(* PLC project LMM.project, Inovance company InoProShop(V1.9.1.6) InoProShop(V1.9.1.6) *)
(* stored: creationDateTime 2026-07-21T20:30:28.2051224, modificationDateTime 2026-07-21T19:55:23.2405761 *)

VAR_GLOBAL  (* GVL *)
  StartBtn AT %IX1.6 : BOOL;  (* 【面板启动】AT %IX1.6 → HMI_xStart/HMI_xEnable（上升沿 STOP→RUN） *)
  StopBtn AT %IX1.4 : BOOL;  (* 【面板停止】AT %IX1.4 → HMI_xStop *)
  ResetBtn : BOOL;  (* 【面板复位】→ HMI_xStopHold3s（错误复位脉冲）；地址现场可另绑 *)
  EStop AT %IX0.4 : BOOL;  (* 【面板急停】AT %IX0.4 正常=TRUE 按下=FALSE → 直通 HMI_xEStop *)
  StopLamp AT %QX0.6 : BOOL;  (* 【停止指示灯】AT %QX0.6 ← Dev_xStop（停止/待机） *)
  StartLamp AT %QX0.7 : BOOL;  (* 【启动/运行指示灯】AT %QX0.7 ← Dev_xRun（正在运行） *)
  JogVel : REAL;  (* 面板点动速度 → 桥接到 HMI_rJogVel* *)
  JogFwd : BOOL;  (* 面板前进 → 按 X 模式映射到 Sync/Diff/独立点动+ *)
  JogBwd : BOOL;  (* 面板后退 → 按 X 模式映射到 Sync/Diff/独立点动- *)
  JogUp : BOOL;  (* 面板上 → HMI_xJogZPos *)
  JogDown : BOOL;  (* 面板下 → HMI_xJogZNeg *)
  JogRight : BOOL;  (* 面板右 → HMI_xJogYPos *)
  JogLeft : BOOL;  (* 面板左 → HMI_xJogYNeg *)
  JogClockAdd : BOOL;  (* 顺时针 *)
  JogClockMis : BOOL;  (* 逆时针 *)
  JogACC : REAL;  (* 点动加速度 → AxisCmd_rAcc *)
  JogDEC : REAL;  (* 点动减速度 → AxisCmd_rDec *)
  HomeReq : BOOL;  (* 面板回零 → HMI_xHomeReqY/Z *)
  CaliForReq : BOOL;  (* 重力标定 *)
  ClearBruch : BOOL;  (* 毛刷清洗 *)
  yLength : REAL;  (* 龙门跨距/Y长度设定 4..6m → HMI_rWheelBase *)
  HMI_xEStop : BOOL;  (* 【急停】TRUE=未按下(正常)；FALSE=急停按下。可按可松，锁存由Logic保持 *)
  HMI_xStop : BOOL;  (* 【设备停止】短按RUN→STOP；长按3s故障复位 *)
  HMI_xStopHold3s : BOOL;  (* 【停止长按满3s脉冲】清急停锁存+轴错误复位+下使能 *)
  HMI_xEnable : BOOL;  (* 【使能/启动别名】与HMI_xStart等效；上升沿STOP→RUN *)
  Dev_xError : BOOL;  (* 【内部故障态】 *)
  Dev_xRun : BOOL;  (* 【内部运行态】 *)
  Dev_xStop : BOOL;  (* 【内部停机态】 *)
  eDevState : INT;  (* 【废弃】不做控制；显示请用 HMI_eDevState 派生 *)
  HMI_xDevError : BOOL;  (* 【故障灯设备级】 *)
  HMI_xDevRun : BOOL;  (* 【运行灯】 *)
  HMI_xDevStop : BOOL;  (* 【停机灯】 *)
  HMI_eOpMode : INT;  (* 【运行方式】0手动 1自动；配合Run灯 *)
  HMI_eDevState : INT;  (* 【设备状态码】0=STOP 1=RUN 2=ERROR *)
  HMI_xStart : BOOL;  (* 【设备启动】瞬时；上升沿STOP→RUN *)
  HMI_xJogYPos : BOOL;  (* 【Y点动+】TRUE移动 FALSE暂停；受限位/Z忙 *)
  HMI_xJogYNeg : BOOL;  (* 【Y点动-】TRUE移动 FALSE暂停 *)
  HMI_xJogZPos : BOOL;  (* 【Z点动+】TRUE移动 FALSE暂停 *)
  HMI_xJogZNeg : BOOL;  (* 【Z点动-】TRUE移动 FALSE暂停 *)
  HMI_xJogRPos : BOOL;  (* 【R点动+】预留；M5未就绪无效 *)
  HMI_xJogRNeg : BOOL;  (* 【R点动-】预留 *)
  HMI_xHomeY : BOOL;  (* 【Y回零】电平/上升沿触发；或配合轴选择 *)
  HMI_xHomeZ : BOOL;  (* 【Z回零】电平/上升沿触发；或配合轴选择 *)
  HMI_xHomeR : BOOL;  (* 【R回零】电平/上升沿触发；或配合轴选择 *)
  HMI_iHomeAxis : INT := 0;  (* 【回零轴选择】0无 1=Y 2=Z 3=R *)
  HMI_xHomeExec : BOOL;  (* 【回零执行】上升沿：对 HMI_iHomeAxis 选定轴启动回零 *)
  HMI_rJogVelX : REAL := 0.4;  (* 【X点动速度】龙门X基速设定 *)
  AxisCmd_rSpinVel : REAL := 0.0;
  HMI_rJogVelR : REAL := 0.2;  (* 【R轴手动速度】 *)
  HMI_rSpinVel : REAL := 0.3;  (* 【X轴旋转速度】 *)
  HMI_rJogVelY : REAL := 0.4;  (* 【Y点动速度】 *)
  HMI_rJogVelZ : REAL := 0.4;  (* 【Z点动速度】 *)
  HMI_rWheelBase : REAL := 5.0;  (* 【龙门跨距=Y行程】单位m，合法范围4..6；自动Y走距用此值 *)
  xEStopLatched : BOOL;  (* 【急停锁存】按下急停置位；仅长按停止复位可清 *)
  xEnablePermit : BOOL;  (* 【废弃】已删除设备态许可互锁 *)
  xFaultAggregate : BOOL;  (* 【故障汇总】任轴Fault *)
  xIlk_BlockYPlus : BOOL;  (* 【联锁禁Y+】由Y+限位派生 *)
  xIlk_BlockYNeg : BOOL;  (* 【联锁禁Y-】由Y-限位派生 *)
  xIlk_BlockZPlus : BOOL;  (* 【联锁禁Z+】由Z+限位派生 *)
  xIlk_BlockZNeg : BOOL;  (* 【联锁禁Z-】由Z-限位派生 *)
  xIlk_BlockYWhenZ : BOOL;  (* 【Z动禁Y】Z运动中禁止Y点动 *)
  xM5Ready : BOOL := TRUE;  (* 【第5轴就绪】TRUE=启用 R(Axis_4)；FALSE=忽略R *)
  HMI_xLampEStop : BOOL;  (* 【急停灯】HMI读；锁存或按钮仍按下 *)
  HMI_xLampEnableOk : BOOL;  (* 【使能/运行灯】=设备RUN *)
  HMI_xLampFault : BOOL;  (* 【轴故障灯】 *)
  eOpMode : INT;  (* 【运行模式】0=手动Manual（本期固定） *)
  iAlarmID : INT;  (* 【内部报警号】Logic判定后拷贝到HMI_iAlarmShow *)
  HMI_iAlarmShow : INT;  (* 【报警号】0无；1001急停；1002故障；1003限位；1004无许可；1099R未就绪 *)
  I_xLimYPos : BOOL;  (* 【Y正限位】物理输入，地址%I* TBD *)
  I_xLimYNeg : BOOL;  (* 【Y负限位】物理输入 *)
  I_xHomeY : BOOL;  (* 【Y原点】物理输入 *)
  I_xLimZPos : BOOL;  (* 【Z正限位】物理输入 *)
  I_xLimZNeg : BOOL;  (* 【Z负限位】物理输入 *)
  I_xHomeZ : BOOL;  (* 【Z原点】物理输入 *)
  I_xLimRPos : BOOL;  (* 【R正限位】预留 *)
  I_xLimRNeg : BOOL;  (* 【R负限位】预留 *)
  I_xHomeR : BOOL;  (* 【R原点】预留 *)
  AxisCmd_xPower : BOOL;  (* 【轴使能命令】仅设备RUN时TRUE *)
  AxisCmd_xJogYPos : BOOL;  (* 【Y点动+命令】含限位/Z忙门控 *)
  AxisCmd_xJogYNeg : BOOL;  (* 【Y点动-命令】 *)
  AxisCmd_xJogZPos : BOOL;  (* 【Z点动+命令】 *)
  AxisCmd_xJogZNeg : BOOL;  (* 【Z点动-命令】 *)
  AxisCmd_xJogRPos : BOOL;  (* 【R点动+命令】预留 *)
  AxisCmd_xJogRNeg : BOOL;  (* 【R点动-命令】预留 *)
  AxisCmd_xHomeY : BOOL;  (* 【Y回零】Logic→Axis；完成/停止后清 *)
  AxisCmd_xHomeZ : BOOL;  (* 【Z回零】Logic→Axis；完成/停止后清 *)
  AxisCmd_xHomeR : BOOL;  (* 【R回零】Logic→Axis；完成/停止后清 *)
  AxisCmd_xStopAll : BOOL;  (* 【全停】急停/停止/故障时TRUE *)
  AxisCmd_xResetFault : BOOL;  (* 【错误复位脉冲】一拍TRUE→各轴MC_Reset *)
  AxisCmd_rWheelBase : REAL;  (* 【跨距L命令】限幅4..6m *)
  AxisCmd_rJogVelX : REAL;  (* 【X点动速度命令】 *)
  AxisCmd_rJogVelY : REAL;  (* 【Y点动速度命令】 *)
  AxisCmd_rJogVelZ : REAL;  (* 【Z点动速度命令】 *)
  AxisCmd_rJogVelR : REAL;  (* 【R点动速度命令】预留 *)
  AxisCmd_rAcc : REAL;  (* 【加速度】 *)
  AxisCmd_rDec : REAL;  (* 【减速度】 *)
  AxisFb_rVelCmdM1 : REAL;  (* 【M1速度指令反馈】供HMI显示 *)
  AxisFb_rVelCmdM2 : REAL;  (* 【M2速度指令反馈】 *)
  AxisFb_rPosM1 : REAL;  (* 【M1实际位置】 *)
  AxisFb_rPosM2 : REAL;  (* 【M2实际位置】 *)
  AxisFb_rPosY : REAL;  (* 【Y实际位置】 *)
  AxisFb_rPosZ : REAL;  (* 【Z实际位置】 *)
  AxisFb_rPosR : REAL;  (* 【R实际位置】预留 *)
  AxisFb_xStandstill1 : BOOL;  (* 【M1静止】 *)
  AxisFb_xStandstill2 : BOOL;  (* 【M2静止】 *)
  AxisFb_xStandstillY : BOOL;  (* 【Y静止】 *)
  AxisFb_xStandstillZ : BOOL;  (* 【Z静止】 *)
  AxisFb_xStandstillR : BOOL;  (* 【R静止】预留 *)
  AxisFb_xMovingM1 : BOOL;  (* 【M1运动中】 *)
  AxisFb_xMovingM2 : BOOL;  (* 【M2运动中】 *)
  AxisFb_xMovingY : BOOL;  (* 【Y运动中】 *)
  AxisFb_xMovingZ : BOOL;  (* 【Z运动中】 *)
  AxisFb_xMovingR : BOOL;  (* 【R运动中】预留 *)
  AxisFb_xPoweredM1 : BOOL;  (* 【M1已使能】驱动功率级就绪，HMI灯 *)
  AxisFb_xPoweredM2 : BOOL;  (* 【M2已使能】 *)
  AxisFb_xPoweredY : BOOL;  (* 【Y已使能】 *)
  AxisFb_xPoweredZ : BOOL;  (* 【Z已使能】 *)
  AxisFb_xPoweredR : BOOL;  (* 【R已使能】预留 *)
  AxisFb_xHomedY : BOOL;  (* 【Y已回零】 *)
  AxisFb_xHomedZ : BOOL;  (* 【Z已回零】 *)
  AxisFb_xHomedR : BOOL;  (* 【R已回零】Axis_4/_MC_Axis[5] *)
  AxisFb_xFaultM1 : BOOL;  (* 【M1故障】 *)
  AxisFb_xFaultM2 : BOOL;  (* 【M2故障】 *)
  AxisFb_xFaultY : BOOL;  (* 【Y故障】 *)
  AxisFb_xFaultZ : BOOL;  (* 【Z故障】 *)
  AxisFb_xFaultR : BOOL;  (* 【R故障】预留 *)
  AxisFb_xReady : BOOL;  (* 【轴就绪】四轴无故障、可参与运动 *)
  HMI_xAutoMode : BOOL;  (* 【自动模式】TRUE自动 FALSE手动 *)
  HMI_xJogXPos : BOOL;  (* 【X+】同步直行 *)
  HMI_xJogXNeg : BOOL;  (* 【X-】 *)
  HMI_xSpinLeft : BOOL;  (* 【左旋转】 *)
  HMI_xSpinRight : BOOL;  (* 【右旋转】 *)
  HMI_xAutoStart : BOOL;  (* 【自动启动】 *)
  HMI_xAutoAbort : BOOL;  (* 【自动中止】 *)
  HMI_rAutoDistX : REAL;  (* 【自动X距离】 *)
  HMI_rAutoVelX : REAL;  (* 【自动X速度】 *)
  HMI_rAutoVelY : REAL;  (* 【自动Y速度】 *)
  HMI_rAutoVelZ : REAL;  (* 【自动Z速度】 *)
  HMI_rForceSet : REAL;  (* 目标力设定(N)，力引导/自动压下用 *)
  HMI_xForceSimEnable : BOOL;  (* 力模拟使能：TRUE用HMI_rForceSim *)
  HMI_rForceSim : REAL;  (* 模拟力设定(N)，仅模拟使能时有效 *)
  HMI_iAutoStepShow : INT;  (* 【自动步号】 *)
  HMI_xAutoBusy : BOOL;  (* 【自动忙】 *)
  HMI_xAutoDone : BOOL;  (* 【自动完成】 *)
  HMI_rForceShow : REAL;  (* 力显示值(N)，供HMI/Web *)
  HMI_xHomedY : BOOL;  (* 【Y已回零】← AxisFb_xHomedY *)
  HMI_xHomedZ : BOOL;  (* 【Z已回零】← AxisFb_xHomedZ *)
  HMI_xHomedR : BOOL;  (* 【R已回零】← AxisFb_xHomedR *)
  HMI_xHomeBusyY : BOOL;  (* 【Y回零中】 *)
  HMI_xHomeBusyZ : BOOL;  (* 【Z回零中】 *)
  HMI_xHomeBusyR : BOOL;  (* 【R回零中】 *)
  Tcp_xConnected : BOOL;  (* 【TCP】已连接 *)
  Tcp_xTimeout : BOOL;  (* 【TCP】通讯超时 *)
  Tcp_xOnline : BOOL;  (* 【TCP】Connected且未超时 *)
  Tcp_xEStop : BOOL := TRUE;  (* 【TCP急停影子】默认TRUE；与面板AND合成 *)
  Tcp_xStop : BOOL;
  Tcp_xStopHold3s : BOOL;
  Tcp_xStart : BOOL;
  Tcp_xEnable : BOOL;
  Tcp_xAutoMode : BOOL;
  Tcp_xJogXPos : BOOL;
  Tcp_xJogXNeg : BOOL;
  Tcp_xSpinLeft : BOOL;
  Tcp_xSpinRight : BOOL;
  Tcp_xJogYPos : BOOL;
  Tcp_xJogYNeg : BOOL;
  Tcp_xJogZPos : BOOL;
  Tcp_xJogZNeg : BOOL;
  Tcp_xJogRPos : BOOL;
  Tcp_xJogRNeg : BOOL;
  Tcp_xHomeY : BOOL;  (* TCP【Y回零】 *)
  Tcp_xHomeZ : BOOL;  (* TCP【Z回零】 *)
  Tcp_xHomeR : BOOL;  (* TCP【R回零】 *)
  Tcp_iHomeAxis : INT := 0;  (* TCP【回零轴选择】0无 1=Y 2=Z 3=R *)
  Tcp_xHomeExec : BOOL;  (* TCP【回零执行】 *)
  Tcp_rJogVelX : REAL := 0.4;
  Tcp_rSpinVel : REAL := 0.3;
  Tcp_rJogVelY : REAL := 0.3;
  Tcp_rJogVelZ : REAL := 0.2;
  Tcp_rJogVelR : REAL := 0.2;
  Tcp_xAutoStart : BOOL;
  Tcp_xAutoAbort : BOOL;
  Tcp_rAutoDistX : REAL := 1.0;
  Tcp_rAutoVelX : REAL := 0.4;
  Tcp_rAutoVelY : REAL := 0.3;
  Tcp_rAutoVelZ : REAL := 0.15;
  Tcp_rWheelBase : REAL := 5.0;
  Tcp_rForceSet : REAL := 100.0;  (* TCP影子：目标力(N) *)
  Tcp_xForceSimEnable : BOOL := TRUE;  (* TCP影子：力模拟使能 *)
  Tcp_rForceSim : REAL;  (* TCP影子：模拟力(N) *)
  Tcp_xForceTare : BOOL;  (* TCP影子：去皮 *)
  Tcp_xForceUntare : BOOL;  (* TCP影子：取消去皮 *)
  Tcp_xForceGuide : BOOL;  (* TCP影子：力引导使能 *)
  Tcp_uiPort : UINT := 9100;  (* 【TCP监听端口】默认9100 *)
  iAutoStep : INT;  (* 【自动步】0Idle..5Done *)
  rForceAct : REAL;  (* 实际力(N)，力传感换算或模拟值 *)
  rForceKp : REAL;  (* 恒力比例增益Kp，力引导Z轴用 *)
  Force_xEnable : BOOL := TRUE;  (* 力传感通讯总使能；FALSE时关闭SM1001 *)
  Force_wInRaw AT %IW102 : WORD;  (* Modbus读通道映射：保持寄存器0x0000原始力值 *)
  Force_xReadTrig : BOOL;  (* 探测读触发；可绑通道上升沿，循环读可不绑 *)
  Force_wOutTare AT %QW42 : WORD;  (* Modbus写通道：寄存器0x0011去皮(1)/取消(2) *)
  Force_wOutUnit AT %QW43 : WORD := 5;  (* Modbus写通道：寄存器0x0002单位，5=牛顿N *)
  Force_rScale : REAL := 0.01;  (* 原始值倍率，默认0.01(百分位) *)
  HMI_xForceTare : BOOL;  (* 去皮触发(上升沿)，面板/外部 *)
  HMI_xForceUntare : BOOL;  (* 取消去皮触发(上升沿) *)
  HMI_xForceGuide : BOOL;  (* 力引导使能：TRUE持续跟力，FALSE停止 *)
  Force_xCommOk : BOOL;  (* 通讯成功(已收到读回文) *)
  Force_xTimeout : BOOL;  (* 通讯超时/失败标志 *)
  Force_xSlaveFail : BOOL;  (* SM1001使能探测失败3次，报警1006 *)
  Force_xTareBusy : BOOL;  (* 去皮命令发送中 *)
  Force_xTareDone : BOOL;  (* 去皮完成脉冲 *)
  Logic_xForceTare : BOOL;  (* 自动步内部去皮脉冲(PRG_Logic写) *)
  Force_iRaw : INT;  (* 有符号原始力计数 *)
  Force_iState : INT;  (* 力任务状态：0闲置1使能2发读3等回文4成功-2失败 *)
  AxisCmd_xJogXPos : BOOL;  (* 【Axis X+】 *)
  AxisCmd_xJogXNeg : BOOL;  (* 【Axis X-】 *)
  AxisCmd_xSpinLeft : BOOL;  (* 【Axis 左旋】 *)
  AxisCmd_xSpinRight : BOOL;  (* 【Axis 右旋】 *)
  AxisCmd_xMoveRelX : BOOL;  (* 【Axis X相对】 *)
  AxisCmd_rMoveDistX : REAL;  (* 【X相对距离】 *)
  AxisCmd_rMoveVelX : REAL;  (* 【X相对速度】 *)
  AxisCmd_xMoveRelY : BOOL;  (* 【Axis Y相对】 *)
  AxisCmd_rMoveDistY : REAL;  (* 【Y相对距离】 *)
  AxisCmd_rMoveVelY : REAL;  (* 【Y相对速度】 *)
  AxisCmd_rZVelCmd : REAL;  (* 【Z速度指令】 *)
  AxisCmd_xUseZVelCmd : BOOL;  (* 【使用Z速度指令】 *)
  AxisCmd_xHoldR : BOOL;  (* 【R保持】 *)
  AxisCmd_rRHoldPos : REAL;  (* 【R保持角】 *)
  AxisFb_xMoveDoneX : BOOL;  (* 【X相对到位】 *)
  AxisFb_xMoveDoneY : BOOL;  (* 【Y相对到位】 *)
END_VAR

PROGRAM PRG_Axis_Control
  VAR
    fbM1 : FB_Servo;
    fbM2 : FB_Servo;
    fbY : FB_Servo;
    fbZ : FB_Servo;
    fbR : FB_Servo;
    fbXDiff : FB_XDiff;
    xPair : BOOL;
    eModeX : INT;
    xDiffPos : BOOL;
    xDiffNeg : BOOL;
    rXVel : REAL;
  END_VAR

            (*==============================================================================
 * PRG_Axis_Control — 运动独立任务（AxisTask）
 * 仅通过 GVL_AxisCmd 输入 / GVL_AxisFb 输出；禁止被外部 CALL
 * 轴绑定：M1=_MC_Axis[1], M2=[2], Y=[3], Z=[4], R=[5]/Axis_4
 *============================================================================*)

(* X：同步直行 / 左右旋；VelX 与 SpinVel 分开 *)
eModeX := 0;
xDiffPos := FALSE; xDiffNeg := FALSE;
IF AxisCmd_xSpinLeft XOR AxisCmd_xSpinRight THEN
	eModeX := 2;
	xDiffPos := AxisCmd_xSpinLeft;
	xDiffNeg := AxisCmd_xSpinRight;
	rXVel := AxisCmd_rSpinVel;
ELSIF AxisCmd_xJogXPos XOR AxisCmd_xJogXNeg THEN
	eModeX := 1;
	rXVel := AxisCmd_rJogVelX;
ELSE
	rXVel := 0.0;
END_IF;

fbXDiff(
	eMode := eModeX,
	eDiffFunc := 1,
	xJogSyncPos := AxisCmd_xJogXPos,
	xJogSyncNeg := AxisCmd_xJogXNeg,
	xJogDiffPos := xDiffPos,
	xJogDiffNeg := xDiffNeg,
	xStop := AxisCmd_xStopAll,
	xEnable := AxisCmd_xPower,
	rJogVel := rXVel,
	rDiffDelta := 0.0,
	rTurnOmega := 0.0,
	rWheelBase := AxisCmd_rWheelBase
);
xPair := fbXDiff.xUsePairVel;

IF xPair THEN
	(* 成对模式：用 FB_XDiff 输出的有符号速度 *)
	fbM1(
		Axis := _MC_Axis[1],
		xEnable := AxisCmd_xPower,
		xJogPos := FALSE, xJogNeg := FALSE,
		xStop := AxisCmd_xStopAll,
		xResetFault := AxisCmd_xResetFault,
		xHome := FALSE,
		xUseVelCmd := TRUE,
		rVelCmd := fbXDiff.rVelCmdM1,
		rJogVel := rXVel,
		rAcc := AxisCmd_rAcc,
		rDec := AxisCmd_rDec
	);
	fbM2(
		Axis := _MC_Axis[2],
		xEnable := AxisCmd_xPower,
		xJogPos := FALSE, xJogNeg := FALSE,
		xStop := AxisCmd_xStopAll,
		xResetFault := AxisCmd_xResetFault,
		xHome := FALSE,
		xUseVelCmd := TRUE,
		rVelCmd := fbXDiff.rVelCmdM2,
		rJogVel := rXVel,
		rAcc := AxisCmd_rAcc,
		rDec := AxisCmd_rDec
	);
	AxisFb_rVelCmdM1 := fbXDiff.rVelCmdM1;
	AxisFb_rVelCmdM2 := fbXDiff.rVelCmdM2;
ELSE
	(* 无 X 命令：两侧保持上电待机 *)
	fbM1(
		Axis := _MC_Axis[1],
		xEnable := AxisCmd_xPower,
		xJogPos := FALSE, xJogNeg := FALSE,
		xStop := AxisCmd_xStopAll,
		xResetFault := AxisCmd_xResetFault,
		xHome := FALSE,
		xUseVelCmd := FALSE,
		rVelCmd := 0.0,
		rJogVel := AxisCmd_rJogVelX,
		rAcc := AxisCmd_rAcc,
		rDec := AxisCmd_rDec
	);
	fbM2(
		Axis := _MC_Axis[2],
		xEnable := AxisCmd_xPower,
		xJogPos := FALSE, xJogNeg := FALSE,
		xStop := AxisCmd_xStopAll,
		xResetFault := AxisCmd_xResetFault,
		xHome := FALSE,
		xUseVelCmd := FALSE,
		rVelCmd := 0.0,
		rJogVel := AxisCmd_rJogVelX,
		rAcc := AxisCmd_rAcc,
		rDec := AxisCmd_rDec
	);
	AxisFb_rVelCmdM1 := 0.0;
	AxisFb_rVelCmdM2 := 0.0;
END_IF;

(* Y / Z / R：回零优先于点动 *)
fbY(
	Axis := _MC_Axis[3],
	xEnable := AxisCmd_xPower,
	xJogPos := AxisCmd_xJogYPos AND NOT AxisCmd_xHomeY,
	xJogNeg := AxisCmd_xJogYNeg AND NOT AxisCmd_xHomeY,
	xStop := AxisCmd_xStopAll,
	xResetFault := AxisCmd_xResetFault,
	xHome := AxisCmd_xHomeY,
	xUseVelCmd := FALSE,
	rVelCmd := 0.0,
	rJogVel := AxisCmd_rJogVelY,
	rAcc := AxisCmd_rAcc,
	rDec := AxisCmd_rDec
);
fbZ(
	Axis := _MC_Axis[4],
	xEnable := AxisCmd_xPower,
	xJogPos := AxisCmd_xJogZPos AND NOT AxisCmd_xUseZVelCmd AND NOT AxisCmd_xHomeZ,
	xJogNeg := AxisCmd_xJogZNeg AND NOT AxisCmd_xUseZVelCmd AND NOT AxisCmd_xHomeZ,
	xStop := AxisCmd_xStopAll,
	xResetFault := AxisCmd_xResetFault,
	xHome := AxisCmd_xHomeZ,
	xUseVelCmd := AxisCmd_xUseZVelCmd AND NOT AxisCmd_xHomeZ,
	rVelCmd := AxisCmd_rZVelCmd,
	rJogVel := AxisCmd_rJogVelZ,
	rAcc := AxisCmd_rAcc,
	rDec := AxisCmd_rDec
);

IF xM5Ready THEN
	fbR(
		Axis := _MC_Axis[5],
		xEnable := AxisCmd_xPower,
		xJogPos := AxisCmd_xJogRPos AND NOT AxisCmd_xHomeR,
		xJogNeg := AxisCmd_xJogRNeg AND NOT AxisCmd_xHomeR,
		xStop := AxisCmd_xStopAll,
		xResetFault := AxisCmd_xResetFault,
		xHome := AxisCmd_xHomeR,
		xUseVelCmd := FALSE,
		rVelCmd := 0.0,
		rJogVel := AxisCmd_rJogVelR,
		rAcc := AxisCmd_rAcc,
		rDec := AxisCmd_rDec
	);
	AxisFb_rPosR := fbR.rActPos;
	AxisFb_xMovingR := fbR.xMoving;
	AxisFb_xPoweredR := fbR.xPowered;
	AxisFb_xFaultR := fbR.xFault;
	AxisFb_xHomedR := fbR.xHomed;
	AxisFb_xStandstillR := fbR.xStandstill;
ELSE
	fbR(
		Axis := _MC_Axis[5],
		xEnable := FALSE,
		xJogPos := FALSE, xJogNeg := FALSE,
		xStop := TRUE,
		xResetFault := FALSE,
		xHome := FALSE,
		xUseVelCmd := FALSE,
		rVelCmd := 0.0,
		rJogVel := 0.0,
		rAcc := AxisCmd_rAcc,
		rDec := AxisCmd_rDec
	);
	AxisFb_xFaultR := FALSE;
	AxisFb_xHomedR := FALSE;
	AxisFb_xMovingR := FALSE;
	AxisFb_xPoweredR := FALSE;
END_IF;

(* ---------- 写反馈区（仅本任务可写） ---------- *)
AxisFb_rPosM1 := fbM1.rActPos;
AxisFb_rPosM2 := fbM2.rActPos;
AxisFb_rPosY := fbY.rActPos;
AxisFb_rPosZ := fbZ.rActPos;
AxisFb_xMovingM1 := fbM1.xMoving;
AxisFb_xMovingM2 := fbM2.xMoving;
AxisFb_xMovingY := fbY.xMoving;
AxisFb_xMovingZ := fbZ.xMoving;
AxisFb_xPoweredM1 := fbM1.xPowered;
AxisFb_xPoweredM2 := fbM2.xPowered;
AxisFb_xPoweredY := fbY.xPowered;
AxisFb_xPoweredZ := fbZ.xPowered;
AxisFb_xFaultM1 := fbM1.xFault;
AxisFb_xFaultM2 := fbM2.xFault;
AxisFb_xFaultY := fbY.xFault;
AxisFb_xFaultZ := fbZ.xFault;
AxisFb_xHomedY := fbY.xHomed;
AxisFb_xHomedZ := fbZ.xHomed;
AxisFb_xStandstill1 := fbM1.xStandstill;
AxisFb_xStandstill2 := fbM2.xStandstill;
AxisFb_xStandstillY := fbY.xStandstill;
AxisFb_xStandstillZ := fbZ.xStandstill;
AxisFb_xReady := NOT (fbM1.xFault OR fbM2.xFault OR fbY.xFault OR fbZ.xFault
	OR (xM5Ready AND AxisFb_xFaultR));

          
END_PROGRAM

FUNCTION_BLOCK FB_TCPServer
  VAR_INPUT
    i_xEnable : BOOL;
    i_uiPort : UINT;
    i_xSendTrig : BOOL;
    i_strSend : STRING(512);
  END_VAR
  VAR_OUTPUT
    o_xConnected : BOOL;
    o_xRecvNew : BOOL;
    o_strRecv : STRING(512);
    o_uiRecvLen : UINT;
    o_xSendDone : BOOL;
    o_xError : BOOL;
    o_wErrorID : WORD;
  END_VAR
  VAR
    SktTCPServer : SktTCPServer;
    SktTCPSend : SktTCPSend;
    SktTCPRecv : SktTCPRecv;
    SktTCPGetStatus : SktTCPGetStatus;
    SktClose : SktClose;
    strLocalAddress : ADDRESS;
    stConnectInfo : CONNECT_INFO;
    diConnectID : CONNECT_ID;
    DataBuffer : ARRAY[1..8192] OF BYTE;  (* 手册样例 ARRAY[1..8192] OF BYTE；abyData:=DataBuffer[1] *)
    R_TRIG_0 : R_TRIG;
    F_TRIG_0 : F_TRIG;
    status : WORD := 0;
    xSendExec : BOOL;
    uiSendSize : UINT;
    i : INT;
    n : INT;
    sOne : STRING(1);
    eStatus : TCP_STATUS;
  END_VAR

            (*==============================================================================
 TCP 服务
 *============================================================================*)
o_xRecvNew := FALSE;
o_xSendDone := FALSE;
o_xConnected := FALSE;

R_TRIG_0(CLK := i_xEnable);
F_TRIG_0(CLK := i_xEnable);

IF R_TRIG_0.Q THEN
	status := 1;
END_IF;

IF F_TRIG_0.Q THEN
	IF (status = 1) OR (status = 2) THEN
		status := 255;
	ELSIF status = 3 THEN
		status := 4;
	END_IF;
END_IF;

CASE status OF
	1: (* 参数初始化 — 手册 *)
		strLocalAddress.strIPAddr := '0.0.0.0';
		strLocalAddress.uiPort := i_uiPort;
		IF strLocalAddress.uiPort < 2000 THEN
			strLocalAddress.uiPort := 9100;
		END_IF;
		diConnectID := 1;
		xSendExec := FALSE;
		uiSendSize := 0;
		status := 2;

	2: (* 创建 TCP Server — 手册 *)
		SktTCPServer(
			xExecute := TRUE,
			diConnectID := diConnectID,
			strLocalAddress := strLocalAddress,
			xDone => ,
			xBusy => ,
			xError => o_xError,
			wErrorID => o_wErrorID,
			stConnectInfo => stConnectInfo);
		IF SktTCPServer.xDone THEN
			status := 3;
		ELSIF SktTCPServer.xError THEN
			status := 255;
		END_IF;

	3: (* 收发 + GetStatus — 手册；ID 用 stConnectInfo.diConnectID *)
		SktTCPGetStatus(
			xEnable := TRUE,
			diConnectID := stConnectInfo.diConnectID,
			xDone => ,
			xBusy => ,
			xError => ,
			wErrorID => ,
			eStatus => eStatus,
			stConnectInfo => );
		IF SktTCPGetStatus.xError THEN
			status := 4;
		ELSIF eStatus <> TCP_STATUS.TCP_ESTABLISHED THEN
			status := 4;
		ELSE
			o_xConnected := TRUE;
			(* Recv：uiDataSize=0 标准模式；abyData:=DataBuffer[1] *)
			SktTCPRecv(
				xEnable := TRUE,
				diConnectID := stConnectInfo.diConnectID,
				abyData := DataBuffer[1],
				uiDataSize := 0,
				xDone => ,
				xBusy => ,
				xError => ,
				wErrorID => ,
				xReady => ,
				uiCount => );
			IF SktTCPRecv.xError THEN
				status := 4;
			ELSIF SktTCPRecv.xDone AND NOT SktTCPRecv.xError THEN
				status := 255;
			ELSE
				(* 有数据：BYTE → JSON 行 STRING *)
				IF SktTCPRecv.xReady AND (SktTCPRecv.uiCount > 0) THEN
					o_xRecvNew := TRUE;
					o_uiRecvLen := SktTCPRecv.uiCount;
					IF o_uiRecvLen > 512 THEN
						n := 512;
					ELSE
						n := UINT_TO_INT(o_uiRecvLen);
					END_IF;
					o_strRecv := '';
					FOR i := 1 TO n DO
						IF (DataBuffer[i] = 16#0A) OR (DataBuffer[i] = 16#0D) THEN
							EXIT;
						END_IF;
						sOne := ' ';
						sOne[1] := DataBuffer[i];
						o_strRecv := CONCAT(o_strRecv, sOne);
					END_FOR;
				END_IF;
				(* 发送：业务触发（非手册 echo） *)
				IF i_xSendTrig AND NOT xSendExec AND (LEN(i_strSend) > 0) THEN
					uiSendSize := INT_TO_UINT(LEN(i_strSend));
					IF uiSendSize > 512 THEN
						uiSendSize := 512;
					END_IF;
					n := UINT_TO_INT(uiSendSize);
					FOR i := 1 TO n DO
						DataBuffer[i] := i_strSend[i];
					END_FOR;
					xSendExec := TRUE;
				END_IF;
				SktTCPSend(
					xExecute := xSendExec,
					diConnectID := stConnectInfo.diConnectID,
					abyData := DataBuffer[1],
					uiDataSize := uiSendSize,
					uiTimeOut := 500,
					xDone => ,
					xBusy => ,
					xError => ,
					wErrorID => );
				IF SktTCPSend.xError THEN
					status := 4;
				ELSIF SktTCPSend.xDone THEN
					SktTCPSend(
						xExecute := FALSE,
						diConnectID := stConnectInfo.diConnectID,
						abyData := DataBuffer[1],
						uiDataSize := 0,
						uiTimeOut := 500,
						xDone => ,
						xBusy => ,
						xError => ,
						wErrorID => );
					xSendExec := FALSE;
					uiSendSize := 0;
					o_xSendDone := TRUE;
				END_IF;
			END_IF;
		END_IF;

	4: (* 关闭 — 手册 SktClose *)
		SktClose(
			xExecute := TRUE,
			diConnectID := stConnectInfo.diConnectID,
			xDone => ,
			xBusy => ,
			xError => ,
			wErrorID => );
		IF SktClose.xDone THEN
			status := 255;
		END_IF;

	255: (* 复位各指令 — 手册 *)
		SktClose(xExecute := FALSE, diConnectID := stConnectInfo.diConnectID, xDone => , xBusy => , xError => , wErrorID => );
		SktTCPSend(xExecute := FALSE, diConnectID := stConnectInfo.diConnectID, abyData := DataBuffer[1], uiDataSize := 0, uiTimeOut := 500, xDone => , xBusy => , xError => , wErrorID => );
		SktTCPRecv(xEnable := FALSE, diConnectID := stConnectInfo.diConnectID, abyData := DataBuffer[1], uiDataSize := 0, xDone => , xBusy => , xError => , wErrorID => , xReady => , uiCount => );
		SktTCPGetStatus(xEnable := FALSE, diConnectID := stConnectInfo.diConnectID, xDone => , xBusy => , xError => , wErrorID => , eStatus => , stConnectInfo => );
		SktTCPServer(xExecute := FALSE, diConnectID := diConnectID, strLocalAddress := strLocalAddress, xDone => , xBusy => , xError => , wErrorID => , stConnectInfo => );
		xSendExec := FALSE;
		o_xError := FALSE;
		(* 仍使能则回到等待下一客户端 *)
		IF i_xEnable THEN
			status := 1;
		END_IF;

ELSE
	;
END_CASE;

          
END_FUNCTION_BLOCK

PROGRAM PRG_TcpHmi
  VAR
    fbTcp : FB_TCPServer;
    tonWatch : TON;
    tonSend : TON;
    abySend : ARRAY[0..1023] OF BYTE;
    abyRecv : ARRAY[0..1023] OF BYTE;
    strLine : STRING(512);
    strOut : STRING(512);
    i : INT;
    n : INT;
    xSendTrig : BOOL;
    uiSendLen : UINT;
    p : INT;
    xInit : BOOL;
  END_VAR

            (*==============================================================================
 * PRG_TcpHmi — TCP JSON HMI 桥（Server :Tcp_uiPort）
 * 写影子 Tcp_*；读 HMI_Status / AxisFb 组 t:s
 *============================================================================*)
IF NOT xInit THEN
	Tcp_xEStop := TRUE;
	Tcp_rJogVelX := 0.4; Tcp_rSpinVel := 0.3;
	Tcp_rJogVelY := 0.3; Tcp_rJogVelZ := 0.2; Tcp_rJogVelR := 0.2;
	Tcp_rAutoDistX := 1.0; Tcp_rAutoVelX := 0.4;
	Tcp_rAutoVelY := 0.3; Tcp_rAutoVelZ := 0.15;
	Tcp_rWheelBase := 5.0; Tcp_rForceSet := 100.0;
	Tcp_xForceSimEnable := TRUE;
	IF Tcp_uiPort = 0 THEN Tcp_uiPort := 9100; END_IF;
	xInit := TRUE;
END_IF;

fbTcp(
	i_xEnable := TRUE,
	i_uiPort := Tcp_uiPort,
	i_xSendTrig := xSendTrig,
	i_strSend := strOut,
	o_xConnected => Tcp_xConnected,
	o_xRecvNew => ,
	o_strRecv => strLine,
	o_uiRecvLen => ,
	o_xSendDone => ,
	o_xError => ,
	o_wErrorID => );

xSendTrig := FALSE;

IF fbTcp.o_xRecvNew THEN
	(* 心跳 *)
	IF FIND(strLine, '"t":"ping"') > 0 OR FIND(strLine, '"t": "ping"') > 0 THEN
		(* pong 随下次状态发 *)
	END_IF;
	(* BOOL *)
	IF FIND(strLine, '"HMI_xEStop":false') > 0 OR FIND(strLine, '"HMI_xEStop": false') > 0 THEN Tcp_xEStop := FALSE;
	ELSIF FIND(strLine, '"HMI_xEStop":true') > 0 OR FIND(strLine, '"HMI_xEStop": true') > 0 THEN Tcp_xEStop := TRUE; END_IF;
	IF FIND(strLine, '"HMI_xStop":true') > 0 THEN Tcp_xStop := TRUE;
	ELSIF FIND(strLine, '"HMI_xStop":false') > 0 THEN Tcp_xStop := FALSE; END_IF;
	IF FIND(strLine, '"HMI_xStopHold3s":true') > 0 THEN Tcp_xStopHold3s := TRUE;
	ELSIF FIND(strLine, '"HMI_xStopHold3s":false') > 0 THEN Tcp_xStopHold3s := FALSE; END_IF;
	IF FIND(strLine, '"HMI_xStart":true') > 0 THEN Tcp_xStart := TRUE; Tcp_xEnable := TRUE;
	ELSIF FIND(strLine, '"HMI_xStart":false') > 0 THEN Tcp_xStart := FALSE; Tcp_xEnable := FALSE; END_IF;
	IF FIND(strLine, '"HMI_xEnable":true') > 0 THEN Tcp_xEnable := TRUE;
	ELSIF FIND(strLine, '"HMI_xEnable":false') > 0 THEN Tcp_xEnable := FALSE; END_IF;
	IF FIND(strLine, '"HMI_xAutoMode":true') > 0 THEN Tcp_xAutoMode := TRUE;
	ELSIF FIND(strLine, '"HMI_xAutoMode":false') > 0 THEN Tcp_xAutoMode := FALSE; END_IF;
	IF FIND(strLine, '"HMI_xJogXPos":true') > 0 THEN Tcp_xJogXPos := TRUE;
	ELSIF FIND(strLine, '"HMI_xJogXPos":false') > 0 THEN Tcp_xJogXPos := FALSE; END_IF;
	IF FIND(strLine, '"HMI_xJogXNeg":true') > 0 THEN Tcp_xJogXNeg := TRUE;
	ELSIF FIND(strLine, '"HMI_xJogXNeg":false') > 0 THEN Tcp_xJogXNeg := FALSE; END_IF;
	IF FIND(strLine, '"HMI_xSpinLeft":true') > 0 THEN Tcp_xSpinLeft := TRUE;
	ELSIF FIND(strLine, '"HMI_xSpinLeft":false') > 0 THEN Tcp_xSpinLeft := FALSE; END_IF;
	IF FIND(strLine, '"HMI_xSpinRight":true') > 0 THEN Tcp_xSpinRight := TRUE;
	ELSIF FIND(strLine, '"HMI_xSpinRight":false') > 0 THEN Tcp_xSpinRight := FALSE; END_IF;
	IF FIND(strLine, '"HMI_xJogYPos":true') > 0 THEN Tcp_xJogYPos := TRUE;
	ELSIF FIND(strLine, '"HMI_xJogYPos":false') > 0 THEN Tcp_xJogYPos := FALSE; END_IF;
	IF FIND(strLine, '"HMI_xJogYNeg":true') > 0 THEN Tcp_xJogYNeg := TRUE;
	ELSIF FIND(strLine, '"HMI_xJogYNeg":false') > 0 THEN Tcp_xJogYNeg := FALSE; END_IF;
	IF FIND(strLine, '"HMI_xJogZPos":true') > 0 THEN Tcp_xJogZPos := TRUE;
	ELSIF FIND(strLine, '"HMI_xJogZPos":false') > 0 THEN Tcp_xJogZPos := FALSE; END_IF;
	IF FIND(strLine, '"HMI_xJogZNeg":true') > 0 THEN Tcp_xJogZNeg := TRUE;
	ELSIF FIND(strLine, '"HMI_xJogZNeg":false') > 0 THEN Tcp_xJogZNeg := FALSE; END_IF;
	IF FIND(strLine, '"HMI_xJogRPos":true') > 0 THEN Tcp_xJogRPos := TRUE;
	ELSIF FIND(strLine, '"HMI_xJogRPos":false') > 0 THEN Tcp_xJogRPos := FALSE; END_IF;
	IF FIND(strLine, '"HMI_xJogRNeg":true') > 0 THEN Tcp_xJogRNeg := TRUE;
	ELSIF FIND(strLine, '"HMI_xJogRNeg":false') > 0 THEN Tcp_xJogRNeg := FALSE; END_IF;
	IF FIND(strLine, '"HMI_xAutoStart":true') > 0 THEN Tcp_xAutoStart := TRUE;
	ELSIF FIND(strLine, '"HMI_xAutoStart":false') > 0 THEN Tcp_xAutoStart := FALSE; END_IF;
	IF FIND(strLine, '"HMI_xAutoAbort":true') > 0 THEN Tcp_xAutoAbort := TRUE;
	ELSIF FIND(strLine, '"HMI_xAutoAbort":false') > 0 THEN Tcp_xAutoAbort := FALSE; END_IF;
	IF FIND(strLine, '"HMI_xForceSimEnable":true') > 0 THEN Tcp_xForceSimEnable := TRUE;
	ELSIF FIND(strLine, '"HMI_xForceSimEnable":false') > 0 THEN Tcp_xForceSimEnable := FALSE; END_IF;
	IF FIND(strLine, '"HMI_xForceTare":true') > 0 THEN Tcp_xForceTare := TRUE;
	ELSIF FIND(strLine, '"HMI_xForceTare":false') > 0 THEN Tcp_xForceTare := FALSE; END_IF;
	IF FIND(strLine, '"HMI_xForceUntare":true') > 0 THEN Tcp_xForceUntare := TRUE;
	ELSIF FIND(strLine, '"HMI_xForceUntare":false') > 0 THEN Tcp_xForceUntare := FALSE; END_IF;
	IF FIND(strLine, '"HMI_xForceGuide":true') > 0 THEN Tcp_xForceGuide := TRUE;
	ELSIF FIND(strLine, '"HMI_xForceGuide":false') > 0 THEN Tcp_xForceGuide := FALSE; END_IF;
	(* REAL：网关保证无空格；键后直接数字 *)
	p := FIND(strLine, '"HMI_rJogVelX":');
	IF p > 0 THEN Tcp_rJogVelX := STRING_TO_REAL(MID(strLine, p + 15, 16)); END_IF;
	p := FIND(strLine, '"HMI_rSpinVel":');
	IF p > 0 THEN Tcp_rSpinVel := STRING_TO_REAL(MID(strLine, p + 14, 16)); END_IF;
	p := FIND(strLine, '"HMI_rJogVelY":');
	IF p > 0 THEN Tcp_rJogVelY := STRING_TO_REAL(MID(strLine, p + 15, 16)); END_IF;
	p := FIND(strLine, '"HMI_rJogVelZ":');
	IF p > 0 THEN Tcp_rJogVelZ := STRING_TO_REAL(MID(strLine, p + 15, 16)); END_IF;
	p := FIND(strLine, '"HMI_rJogVelR":');
	IF p > 0 THEN Tcp_rJogVelR := STRING_TO_REAL(MID(strLine, p + 15, 16)); END_IF;
	p := FIND(strLine, '"HMI_rAutoDistX":');
	IF p > 0 THEN Tcp_rAutoDistX := STRING_TO_REAL(MID(strLine, p + 16, 16)); END_IF;
	p := FIND(strLine, '"HMI_rAutoVelX":');
	IF p > 0 THEN Tcp_rAutoVelX := STRING_TO_REAL(MID(strLine, p + 15, 16)); END_IF;
	p := FIND(strLine, '"HMI_rAutoVelY":');
	IF p > 0 THEN Tcp_rAutoVelY := STRING_TO_REAL(MID(strLine, p + 15, 16)); END_IF;
	p := FIND(strLine, '"HMI_rAutoVelZ":');
	IF p > 0 THEN Tcp_rAutoVelZ := STRING_TO_REAL(MID(strLine, p + 15, 16)); END_IF;
	p := FIND(strLine, '"HMI_rWheelBase":');
	IF p > 0 THEN Tcp_rWheelBase := STRING_TO_REAL(MID(strLine, p + 16, 16)); END_IF;
	p := FIND(strLine, '"HMI_rForceSet":');
	IF p > 0 THEN Tcp_rForceSet := STRING_TO_REAL(MID(strLine, p + 15, 16)); END_IF;
	p := FIND(strLine, '"HMI_rForceSim":');
	IF p > 0 THEN Tcp_rForceSim := STRING_TO_REAL(MID(strLine, p + 15, 16)); END_IF;
END_IF;

(* 有接收则本周期 IN=FALSE 复位；否则连接中计时 *)
tonWatch(IN := Tcp_xConnected AND NOT fbTcp.o_xRecvNew, PT := T#500MS);
Tcp_xTimeout := Tcp_xConnected AND tonWatch.Q;
IF Tcp_xTimeout OR NOT Tcp_xConnected THEN
	Tcp_xStop := FALSE; Tcp_xStopHold3s := FALSE;
	Tcp_xStart := FALSE; Tcp_xEnable := FALSE;
	Tcp_xJogXPos := FALSE; Tcp_xJogXNeg := FALSE;
	Tcp_xSpinLeft := FALSE; Tcp_xSpinRight := FALSE;
	Tcp_xJogYPos := FALSE; Tcp_xJogYNeg := FALSE;
	Tcp_xJogZPos := FALSE; Tcp_xJogZNeg := FALSE;
	Tcp_xJogRPos := FALSE; Tcp_xJogRNeg := FALSE;
	Tcp_xAutoStart := FALSE; Tcp_xAutoAbort := FALSE;
	Tcp_xForceTare := FALSE; Tcp_xForceUntare := FALSE;
	IF Tcp_xTimeout OR NOT Tcp_xConnected THEN Tcp_xEStop := TRUE; END_IF;
END_IF;

tonSend(IN := NOT tonSend.Q, PT := T#100MS);
IF tonSend.Q AND Tcp_xConnected THEN
	strOut := '{"t":"s"';
	strOut := CONCAT(strOut, ',"HMI_eDevState":');
	strOut := CONCAT(strOut, INT_TO_STRING(HMI_eDevState));
	strOut := CONCAT(strOut, ',"HMI_eOpMode":');
	strOut := CONCAT(strOut, INT_TO_STRING(HMI_eOpMode));
	strOut := CONCAT(strOut, ',"HMI_iAutoStepShow":');
	strOut := CONCAT(strOut, INT_TO_STRING(HMI_iAutoStepShow));
	strOut := CONCAT(strOut, ',"HMI_iAlarmShow":');
	strOut := CONCAT(strOut, INT_TO_STRING(HMI_iAlarmShow));
	strOut := CONCAT(strOut, ',"HMI_xDevStop":');
	strOut := CONCAT(strOut, SEL(HMI_xDevStop, 'false', 'true'));
	strOut := CONCAT(strOut, ',"HMI_xDevRun":');
	strOut := CONCAT(strOut, SEL(HMI_xDevRun, 'false', 'true'));
	strOut := CONCAT(strOut, ',"HMI_xDevError":');
	strOut := CONCAT(strOut, SEL(HMI_xDevError, 'false', 'true'));
	strOut := CONCAT(strOut, ',"HMI_xAutoBusy":');
	strOut := CONCAT(strOut, SEL(HMI_xAutoBusy, 'false', 'true'));
	strOut := CONCAT(strOut, ',"HMI_xAutoDone":');
	strOut := CONCAT(strOut, SEL(HMI_xAutoDone, 'false', 'true'));
	strOut := CONCAT(strOut, ',"HMI_xLampEStop":');
	strOut := CONCAT(strOut, SEL(HMI_xLampEStop, 'false', 'true'));
	strOut := CONCAT(strOut, ',"HMI_xLampEnableOk":');
	strOut := CONCAT(strOut, SEL(HMI_xLampEnableOk, 'false', 'true'));
	strOut := CONCAT(strOut, ',"HMI_xLampFault":');
	strOut := CONCAT(strOut, SEL(HMI_xLampFault, 'false', 'true'));
	strOut := CONCAT(strOut, ',"HMI_rForceShow":');
	strOut := CONCAT(strOut, REAL_TO_STRING(HMI_rForceShow));
	strOut := CONCAT(strOut, ',"Force_xCommOk":');
	strOut := CONCAT(strOut, SEL(Force_xCommOk, 'false', 'true'));
	strOut := CONCAT(strOut, ',"Force_xTareBusy":');
	strOut := CONCAT(strOut, SEL(Force_xTareBusy, 'false', 'true'));
	strOut := CONCAT(strOut, ',"Force_xTareDone":');
	strOut := CONCAT(strOut, SEL(Force_xTareDone, 'false', 'true'));
	strOut := CONCAT(strOut, ',"HMI_xForceGuide":');
	strOut := CONCAT(strOut, SEL(HMI_xForceGuide, 'false', 'true'));
	strOut := CONCAT(strOut, ',"Force_xSlaveFail":');
	strOut := CONCAT(strOut, SEL(Force_xSlaveFail, 'false', 'true'));
	strOut := CONCAT(strOut, ',"Tcp_xConnected":true,"Tcp_xTimeout":');
	strOut := CONCAT(strOut, SEL(Tcp_xTimeout, 'false', 'true'));
	strOut := CONCAT(strOut, ',"AxisFb_rPosY":');
	strOut := CONCAT(strOut, REAL_TO_STRING(AxisFb_rPosY));
	strOut := CONCAT(strOut, ',"AxisFb_rPosZ":');
	strOut := CONCAT(strOut, REAL_TO_STRING(AxisFb_rPosZ));
	strOut := CONCAT(strOut, ',"AxisFb_xReady":');
	strOut := CONCAT(strOut, SEL(AxisFb_xReady, 'false', 'true'));
	strOut := CONCAT(strOut, '}');
	strOut := CONCAT(strOut, '$N');
	xSendTrig := TRUE;
END_IF;

          
END_PROGRAM

FUNCTION_BLOCK FB_XDiff
  VAR_INPUT
    eMode : INT;
    eDiffFunc : INT;
    xJogSyncPos : BOOL;
    xJogSyncNeg : BOOL;
    xJogDiffPos : BOOL;
    xJogDiffNeg : BOOL;
    xStop : BOOL;
    xEnable : BOOL;
    rJogVel : REAL;
    rDiffDelta : REAL;
    rTurnOmega : REAL;
    rWheelBase : REAL;
  END_VAR
  VAR_OUTPUT
    rVelCmdM1 : REAL;
    rVelCmdM2 : REAL;
    xActive : BOOL;
    xUsePairVel : BOOL;
    xWheelBaseOk : BOOL;
  END_VAR

            (*==============================================================================
 * FB_XDiff — 龙门 X 双驱速度合成（仅 Axis 任务内使用）
 * eMode: 0=独立  1=同步同速平移  2=差速（子功能见 eDiffFunc）
 * eDiffFunc: 0=纠偏  1=原地旋转(一正一反)  2=差速拐弯
 * 跨距 rWheelBase: 4..6 m；X 运动方向与 Y 垂直
 *============================================================================*)

(* 输出清零 *)
rVelCmdM1 := 0.0;
rVelCmdM2 := 0.0;
xUsePairVel := FALSE;
xActive := FALSE;
(* 跨距合法性 *)
xWheelBaseOk := (rWheelBase >= 4.0) AND (rWheelBase <= 6.0);

(* 未使能 / 停止 / 独立模式：不合成成对速度 *)
IF NOT xEnable OR xStop OR eMode = 0 THEN
	RETURN;
END_IF;

(* ---------- Sync：两侧同速，龙门沿 X 平移 ---------- *)
IF eMode = 1 THEN
	IF xJogSyncPos XOR xJogSyncNeg THEN
		xUsePairVel := TRUE;
		xActive := TRUE;
		IF xJogSyncPos THEN
			rVelCmdM1 := rJogVel;
		ELSE
			rVelCmdM1 := -rJogVel;
		END_IF;
		rVelCmdM2 := rVelCmdM1; (* 同速 *)
	END_IF;
	RETURN;
END_IF;

(* ---------- Diff：需有方向键 ---------- *)
IF NOT (xJogDiffPos XOR xJogDiffNeg) THEN
	RETURN;
END_IF;

(* 原地旋转 / 差速拐弯依赖合法跨距 *)
IF (eDiffFunc = 1 OR eDiffFunc = 2) AND NOT xWheelBaseOk THEN
	RETURN;
END_IF;

xUsePairVel := TRUE;
xActive := TRUE;

CASE eDiffFunc OF
	0: (* 纠偏：同向 V±Δ，扶正龙门 *)
		IF xJogDiffPos THEN
			rVelCmdM1 := rJogVel + rDiffDelta;
			rVelCmdM2 := rJogVel - rDiffDelta;
		ELSE
			rVelCmdM1 := -(rJogVel + rDiffDelta);
			rVelCmdM2 := -(rJogVel - rDiffDelta);
		END_IF;

	1: (* 原地旋转：M1/M2 一正一反，转角度 *)
		IF ABS(rTurnOmega) > 1.0E-6 THEN
			rVelCmdM1 := rTurnOmega * rWheelBase * 0.5;
		ELSE
			rVelCmdM1 := rJogVel;
		END_IF;
		rVelCmdM2 := -rVelCmdM1;
		IF xJogDiffNeg THEN
			rVelCmdM1 := -rVelCmdM1;
			rVelCmdM2 := -rVelCmdM2;
		END_IF;

	2: (* 差速拐弯：两侧同向为主，速度差，可边走边弯 *)
		IF ABS(rTurnOmega) > 1.0E-6 THEN
			rVelCmdM1 := rJogVel + rTurnOmega * rWheelBase * 0.5;
			rVelCmdM2 := rJogVel - rTurnOmega * rWheelBase * 0.5;
		ELSE
			rVelCmdM1 := rJogVel + rDiffDelta;
			rVelCmdM2 := rJogVel - rDiffDelta;
		END_IF;
		IF xJogDiffNeg THEN
			rVelCmdM1 := -rVelCmdM1;
			rVelCmdM2 := -rVelCmdM2;
		END_IF;

ELSE
	xUsePairVel := FALSE;
	xActive := FALSE;
END_CASE;

          
END_FUNCTION_BLOCK

PROGRAM PLC_PRG

            (*==============================================================================
 * PLC_PRG — 主任务入口（MainTask）
 * SM1001 由 PRG_Force485 管理；禁止在此 CALL PRG_Axis_Control
 *============================================================================*)
PRG_Force485();
PRG_TcpHmi();
PRG_Logic();

          
END_PROGRAM

PROGRAM PRG_Logic
  VAR
    tonHold : TON;
    xResetPulse : BOOL;
    xResetPrev : BOOL;
    xSafe : BOOL;
    xAutoStartPrev : BOOL;
    xAutoStartEdge : BOOL;
    rRHold : REAL;
    xMoveXSent : BOOL;
    xMoveYSent : BOOL;
    xGuidePrev : BOOL;
    xAutoTareSent : BOOL;
    xDoForceFollow : BOOL;
    xBridgeInited : BOOL;
    xHomeTrigY : BOOL;
    xHomeTrigZ : BOOL;
    xHomeTrigR : BOOL;
    xHomeTrigYPrev : BOOL;
    xHomeTrigZPrev : BOOL;
    xHomeTrigRPrev : BOOL;
    xAnyHomeBusy : BOOL;
    eCtrlSrc : INT;  (* 0=面板独占 1=TCP独占 *)
    xPanelAct : BOOL;
    xTcpAct : BOOL;
  END_VAR

            (*==============================================================================
 * PRG_Logic — 精简：无 eDevState
 * 硬条件仅：急停(TRUE正常) + 电机 Errorstop + Y/Z限位
 * 力传感故障只报警，不挡轴
 *============================================================================*)

(* —— 面板 ‖ TCP 并行互斥：谁激活用谁；禁止 OR 混控 / 用 0 盖设定 —— *)
Tcp_xOnline := Tcp_xConnected AND NOT Tcp_xTimeout;

(* 激活检测：本拍有操作请求 *)
xPanelAct := StartBtn OR StopBtn OR ResetBtn
	OR JogFwd OR JogBwd OR JogLeft OR JogRight OR JogUp OR JogDown;
(* 仅操作请求算激活；常驻模式位不算，避免在线就永久抢占 *)
xTcpAct := Tcp_xOnline AND (
	Tcp_xStart OR Tcp_xStop OR Tcp_xStopHold3s OR Tcp_xEnable
	OR Tcp_xJogXPos OR Tcp_xJogXNeg OR Tcp_xSpinLeft OR Tcp_xSpinRight
	OR Tcp_xJogYPos OR Tcp_xJogYNeg OR Tcp_xJogZPos OR Tcp_xJogZNeg
	OR Tcp_xJogRPos OR Tcp_xJogRNeg
	OR Tcp_xHomeY OR Tcp_xHomeZ OR Tcp_xHomeR OR Tcp_xHomeExec
	OR Tcp_xAutoStart OR Tcp_xAutoAbort
	OR Tcp_xForceGuide OR Tcp_xForceTare OR Tcp_xForceUntare);

IF NOT Tcp_xOnline THEN
	eCtrlSrc := 0;	(* 掉线强制回面板 *)
ELSIF xTcpAct THEN
	eCtrlSrc := 1;
ELSIF xPanelAct THEN
	eCtrlSrc := 0;
END_IF;
(* 双方都闲：保持 eCtrlSrc，设定值不跳变 *)

IF eCtrlSrc = 1 THEN
	(* ===== TCP 独占：整组用 Tcp_* 当前值 ===== *)
	HMI_xStop := Tcp_xStop;
	HMI_xStart := Tcp_xStart;
	HMI_xEnable := Tcp_xEnable OR Tcp_xStart;
	HMI_xStopHold3s := Tcp_xStopHold3s;
	HMI_xAutoMode := Tcp_xAutoMode;
	HMI_xForceSimEnable := Tcp_xForceSimEnable;
	HMI_xForceGuide := Tcp_xForceGuide;
	HMI_xForceTare := Tcp_xForceTare;
	HMI_xForceUntare := Tcp_xForceUntare;
	HMI_xJogXPos := Tcp_xJogXPos;
	HMI_xJogXNeg := Tcp_xJogXNeg;
	HMI_xSpinLeft := Tcp_xSpinLeft;
	HMI_xSpinRight := Tcp_xSpinRight;
	HMI_xJogYPos := Tcp_xJogYPos;
	HMI_xJogYNeg := Tcp_xJogYNeg;
	HMI_xJogZPos := Tcp_xJogZPos;
	HMI_xJogZNeg := Tcp_xJogZNeg;
	HMI_xJogRPos := Tcp_xJogRPos;
	HMI_xJogRNeg := Tcp_xJogRNeg;
	HMI_xHomeY := Tcp_xHomeY;
	HMI_xHomeZ := Tcp_xHomeZ;
	HMI_xHomeR := Tcp_xHomeR;
	HMI_iHomeAxis := Tcp_iHomeAxis;
	HMI_xHomeExec := Tcp_xHomeExec;
	HMI_xAutoStart := Tcp_xAutoStart;
	HMI_xAutoAbort := Tcp_xAutoAbort;
	HMI_rJogVelX := Tcp_rJogVelX;
	HMI_rSpinVel := Tcp_rSpinVel;
	HMI_rJogVelY := Tcp_rJogVelY;
	HMI_rJogVelZ := Tcp_rJogVelZ;
	HMI_rJogVelR := Tcp_rJogVelR;
	HMI_rAutoDistX := Tcp_rAutoDistX;
	HMI_rAutoVelX := Tcp_rAutoVelX;
	HMI_rAutoVelY := Tcp_rAutoVelY;
	HMI_rAutoVelZ := Tcp_rAutoVelZ;
	HMI_rWheelBase := Tcp_rWheelBase;
	HMI_rForceSet := Tcp_rForceSet;
	HMI_rForceSim := Tcp_rForceSim;
ELSE
	(* ===== 面板独占：整组用面板；TCP 数值一律不参与 ===== *)
	HMI_xStop := StopBtn;
	HMI_xStart := StartBtn;
	HMI_xEnable := StartBtn;
	HMI_xStopHold3s := ResetBtn;
	HMI_xJogXPos := JogFwd;
	HMI_xJogXNeg := JogBwd;
	HMI_xSpinLeft := FALSE;
	HMI_xSpinRight := FALSE;
	HMI_xJogYPos := JogRight;
	HMI_xJogYNeg := JogLeft;
	HMI_xJogZPos := JogUp;
	HMI_xJogZNeg := JogDown;
	HMI_xJogRPos := FALSE;
	HMI_xJogRNeg := FALSE;
	HMI_xHomeY := FALSE;
	HMI_xHomeZ := FALSE;
	HMI_xHomeR := FALSE;
	HMI_xHomeExec := FALSE;
	HMI_xAutoStart := FALSE;
	HMI_xAutoAbort := FALSE;
	HMI_xForceGuide := FALSE;
	HMI_xForceTare := FALSE;
	HMI_xForceUntare := FALSE;
	HMI_rJogVelX := JogVel;
	HMI_rJogVelY := JogVel;
	HMI_rJogVelZ := JogVel;
	(* Spin/R/自动/力设定：保持上次 HMI_r*，禁止用 Tcp 默认 0 覆盖 *)
END_IF;

(* 安全叠加：急停双方都正常才放行；停止/中止任一通道可介入 *)
HMI_xEStop := EStop AND Tcp_xEStop;
HMI_xStop := HMI_xStop OR StopBtn OR Tcp_xStop;
HMI_xStopHold3s := HMI_xStopHold3s OR ResetBtn OR Tcp_xStopHold3s;
HMI_xAutoAbort := HMI_xAutoAbort OR Tcp_xAutoAbort;

(* —— 急停锁存 / 长按复位 —— *)
IF NOT HMI_xEStop THEN
	xEStopLatched := TRUE;
END_IF;
tonHold(IN := HMI_xStop AND HMI_xEStop, PT := T#3S);
xResetPulse := (HMI_xStopHold3s OR tonHold.Q) AND NOT xResetPrev;
xResetPrev := HMI_xStopHold3s OR tonHold.Q;
IF xResetPulse THEN
	xEStopLatched := FALSE;
	AxisCmd_xResetFault := TRUE;
	iAutoStep := 0;
	Force_xSlaveFail := FALSE;
ELSE
	AxisCmd_xResetFault := FALSE;
END_IF;

(* 电机报警汇总：仅各轴 ReadStatus.Errorstop *)
xFaultAggregate := AxisFb_xFaultM1 OR AxisFb_xFaultM2 OR AxisFb_xFaultY OR AxisFb_xFaultZ
	OR (xM5Ready AND AxisFb_xFaultR);

IF HMI_xAutoMode THEN
	eOpMode := 1;
ELSE
	eOpMode := 0;
END_IF;
HMI_eOpMode := eOpMode;

(* 安全可运行：急停正常且未锁存 *)
xSafe := HMI_xEStop AND NOT xEStopLatched;

(* 上电：不靠设备态；急停正常即允许 Power *)
AxisCmd_xPower := xSafe;
(* 停止：停止钮 / 急停 / 电机报警 / 自动中止 *)
AxisCmd_xStopAll := HMI_xStop OR NOT xSafe OR xFaultAggregate OR HMI_xAutoAbort;

(* 状态灯：由条件推导，不是状态机 *)
Dev_xError := xFaultAggregate;
Dev_xRun := xSafe AND NOT HMI_xStop AND NOT xFaultAggregate;
Dev_xStop := NOT Dev_xRun AND NOT Dev_xError;
HMI_xDevError := Dev_xError;
HMI_xDevRun := Dev_xRun;
HMI_xDevStop := Dev_xStop;
(* 仅给 HMI/Web 显示用，不参与互锁 *)
IF Dev_xError THEN
	HMI_eDevState := 2;
ELSIF Dev_xRun THEN
	HMI_eDevState := 1;
ELSE
	HMI_eDevState := 0;
END_IF;

IF HMI_xForceSimEnable THEN
	rForceAct := HMI_rForceSim;
END_IF;
HMI_rForceShow := rForceAct;
IF rForceKp < 1.0E-6 THEN
	rForceKp := 1.0;
END_IF;

xIlk_BlockYPlus := I_xLimYPos;
xIlk_BlockYNeg := I_xLimYNeg;
(* Z 回零后软限位写死：[−0.7, 0]；未回零仅硬件限位 *)
xIlk_BlockZPlus := I_xLimZPos
	OR (AxisFb_xHomedZ AND (AxisFb_rPosZ >= 0.0));
xIlk_BlockZNeg := I_xLimZNeg
	OR (AxisFb_xHomedZ AND (AxisFb_rPosZ <= -0.7));

AxisCmd_rJogVelX := HMI_rJogVelX;
AxisCmd_rSpinVel := HMI_rSpinVel;
AxisCmd_rJogVelY := HMI_rJogVelY;
AxisCmd_rJogVelZ := HMI_rJogVelZ;
AxisCmd_rJogVelR := HMI_rJogVelR;
AxisCmd_rWheelBase := LIMIT(4.0, HMI_rWheelBase, 6.0);
AxisCmd_rAcc := JogACC;
AxisCmd_rDec := JogDEC;
IF AxisCmd_rAcc < 1.0 THEN
	AxisCmd_rAcc := 100.0;
END_IF;
IF AxisCmd_rDec < 1.0 THEN
	AxisCmd_rDec := 100.0;
END_IF;

AxisCmd_xJogXPos := FALSE;
AxisCmd_xJogXNeg := FALSE;
AxisCmd_xSpinLeft := FALSE;
AxisCmd_xSpinRight := FALSE;
AxisCmd_xJogYPos := FALSE;
AxisCmd_xJogYNeg := FALSE;
AxisCmd_xJogZPos := FALSE;
AxisCmd_xJogZNeg := FALSE;
AxisCmd_xJogRPos := FALSE;
AxisCmd_xJogRNeg := FALSE;
AxisCmd_xUseZVelCmd := FALSE;
AxisCmd_rZVelCmd := 0.0;
AxisCmd_xMoveRelX := FALSE;
AxisCmd_xMoveRelY := FALSE;
AxisCmd_xHoldR := FALSE;

xAutoStartEdge := HMI_xAutoStart AND NOT xAutoStartPrev;
xAutoStartPrev := HMI_xAutoStart;

IF HMI_xAutoAbort OR NOT xSafe OR xFaultAggregate THEN
	iAutoStep := 0;
	HMI_xAutoBusy := FALSE;
END_IF;

(* ===== 手动：急停正常 + 未按停止 + 手动模式 ===== *)
IF xSafe AND (eOpMode = 0) AND NOT HMI_xStop AND NOT xFaultAggregate THEN
	IF HMI_xSpinLeft XOR HMI_xSpinRight THEN
		AxisCmd_xSpinLeft := HMI_xSpinLeft;
		AxisCmd_xSpinRight := HMI_xSpinRight;
	ELSIF HMI_xJogXPos XOR HMI_xJogXNeg THEN
		AxisCmd_xJogXPos := HMI_xJogXPos;
		AxisCmd_xJogXNeg := HMI_xJogXNeg;
	END_IF;
	AxisCmd_xJogYPos := HMI_xJogYPos AND NOT xIlk_BlockYPlus;
	AxisCmd_xJogYNeg := HMI_xJogYNeg AND NOT xIlk_BlockYNeg;
	AxisCmd_xJogZPos := HMI_xJogZPos AND NOT xIlk_BlockZPlus;
	AxisCmd_xJogZNeg := HMI_xJogZNeg AND NOT xIlk_BlockZNeg;
	IF xM5Ready THEN
		AxisCmd_xJogRPos := HMI_xJogRPos;
		AxisCmd_xJogRNeg := HMI_xJogRNeg;
	END_IF;
END_IF;

(* ===== 自动 ===== *)
IF xSafe AND (eOpMode = 1) AND NOT HMI_xStop AND NOT xFaultAggregate THEN
	IF iAutoStep = 0 AND xAutoStartEdge THEN
		iAutoStep := 1;
		rRHold := AxisFb_rPosR;
		xAutoTareSent := FALSE;
		HMI_xAutoDone := FALSE;
		HMI_xAutoBusy := TRUE;
	END_IF;

	CASE iAutoStep OF
		1:
			AxisCmd_xHoldR := TRUE;
			AxisCmd_rRHoldPos := rRHold;
			AxisCmd_rMoveDistX := HMI_rAutoDistX;
			AxisCmd_rMoveVelX := HMI_rAutoVelX;
			AxisCmd_xMoveRelX := TRUE;
			IF AxisFb_xMoveDoneX THEN
				AxisCmd_xMoveRelX := FALSE;
				xAutoTareSent := FALSE;
				iAutoStep := 2;
			END_IF;
		2:
			IF NOT xAutoTareSent THEN
				Logic_xForceTare := TRUE;
				xAutoTareSent := TRUE;
			END_IF;
			AxisCmd_xHoldR := TRUE;
			AxisCmd_rRHoldPos := rRHold;
			IF rForceAct >= HMI_rForceSet AND HMI_xForceGuide THEN
				iAutoStep := 3;
			END_IF;
		3:
			AxisCmd_xHoldR := TRUE;
			AxisCmd_rRHoldPos := rRHold;
			AxisCmd_rMoveDistY := AxisCmd_rWheelBase;
			AxisCmd_rMoveVelY := HMI_rAutoVelY;
			AxisCmd_xMoveRelY := TRUE;
			IF AxisFb_xMoveDoneY THEN
				AxisCmd_xMoveRelY := FALSE;
				iAutoStep := 4;
			END_IF;
		4:
			iAutoStep := 5;
		5:
			HMI_xAutoBusy := FALSE;
			HMI_xAutoDone := TRUE;
			iAutoStep := 0;
	END_CASE;
END_IF;


(* ===== 回零：轴选择 + 独立触发；Y/Z/R；完成→当前位置=0 ===== *)
xHomeTrigY := HMI_xHomeY OR ((HMI_iHomeAxis = 1) AND HMI_xHomeExec);
xHomeTrigZ := HMI_xHomeZ OR ((HMI_iHomeAxis = 2) AND HMI_xHomeExec);
xHomeTrigR := HMI_xHomeR OR ((HMI_iHomeAxis = 3) AND HMI_xHomeExec);
xAnyHomeBusy := AxisCmd_xHomeY OR AxisCmd_xHomeZ OR AxisCmd_xHomeR;

IF AxisCmd_xStopAll OR NOT xSafe OR xFaultAggregate THEN
	AxisCmd_xHomeY := FALSE;
	AxisCmd_xHomeZ := FALSE;
	AxisCmd_xHomeR := FALSE;
ELSE
	(* 回零完成：清命令 *)
	IF AxisCmd_xHomeY AND AxisFb_xHomedY THEN
		AxisCmd_xHomeY := FALSE;
	END_IF;
	IF AxisCmd_xHomeZ AND AxisFb_xHomedZ THEN
		AxisCmd_xHomeZ := FALSE;
	END_IF;
	IF AxisCmd_xHomeR AND AxisFb_xHomedR THEN
		AxisCmd_xHomeR := FALSE;
	END_IF;

	(* 手动：上升沿启动；同时只回一轴 *)
	IF (eOpMode = 0) AND NOT HMI_xStop THEN
		IF xHomeTrigY AND NOT xHomeTrigYPrev AND NOT xAnyHomeBusy THEN
			AxisCmd_xHomeY := TRUE;
			AxisCmd_xHomeZ := FALSE;
			AxisCmd_xHomeR := FALSE;
		ELSIF xHomeTrigZ AND NOT xHomeTrigZPrev AND NOT xAnyHomeBusy THEN
			AxisCmd_xHomeY := FALSE;
			AxisCmd_xHomeZ := TRUE;
			AxisCmd_xHomeR := FALSE;
		ELSIF xHomeTrigR AND NOT xHomeTrigRPrev AND NOT xAnyHomeBusy AND xM5Ready THEN
			AxisCmd_xHomeY := FALSE;
			AxisCmd_xHomeZ := FALSE;
			AxisCmd_xHomeR := TRUE;
		END_IF;
	END_IF;
END_IF;
xHomeTrigYPrev := xHomeTrigY;
xHomeTrigZPrev := xHomeTrigZ;
xHomeTrigRPrev := xHomeTrigR;

(* 回零中禁止同轴点动（命令侧再挡一层） *)
IF AxisCmd_xHomeY THEN
	AxisCmd_xJogYPos := FALSE;
	AxisCmd_xJogYNeg := FALSE;
END_IF;
IF AxisCmd_xHomeZ THEN
	AxisCmd_xJogZPos := FALSE;
	AxisCmd_xJogZNeg := FALSE;
	AxisCmd_xUseZVelCmd := FALSE;
END_IF;
IF AxisCmd_xHomeR THEN
	AxisCmd_xJogRPos := FALSE;
	AxisCmd_xJogRNeg := FALSE;
END_IF;

HMI_xHomedY := AxisFb_xHomedY;
HMI_xHomedZ := AxisFb_xHomedZ;
HMI_xHomedR := AxisFb_xHomedR;
HMI_xHomeBusyY := AxisCmd_xHomeY;
HMI_xHomeBusyZ := AxisCmd_xHomeZ;
HMI_xHomeBusyR := AxisCmd_xHomeR;

(* ===== 力引导 ===== *)
xDoForceFollow := HMI_xForceGuide AND xSafe AND NOT HMI_xStop AND NOT xFaultAggregate
	AND (HMI_xForceSimEnable OR Force_xCommOk);
IF xDoForceFollow THEN
	IF NOT (HMI_xJogZPos OR HMI_xJogZNeg) THEN
		AxisCmd_xUseZVelCmd := TRUE;
		AxisCmd_rZVelCmd := LIMIT(-ABS(HMI_rAutoVelZ),
			rForceKp * (HMI_rForceSet - rForceAct), ABS(HMI_rAutoVelZ));
		IF ABS(HMI_rForceSet - rForceAct) < 0.5 THEN
			AxisCmd_rZVelCmd := 0.0;
		END_IF;
		(* 力跟随位移限制在回零后软限位 [−0.7, 0] 内 *)
		IF AxisFb_xHomedZ THEN
			IF (AxisFb_rPosZ >= 0.0) AND (AxisCmd_rZVelCmd > 0.0) THEN
				AxisCmd_rZVelCmd := 0.0;
			END_IF;
			IF (AxisFb_rPosZ <= -0.7) AND (AxisCmd_rZVelCmd < 0.0) THEN
				AxisCmd_rZVelCmd := 0.0;
			END_IF;
		END_IF;
	END_IF;
END_IF;

IF xEStopLatched OR NOT HMI_xEStop THEN
	iAlarmID := 1001;
ELSIF xFaultAggregate THEN
	iAlarmID := 1002;
ELSIF NOT HMI_xForceSimEnable AND Force_xSlaveFail THEN
	iAlarmID := 1006;
ELSIF NOT HMI_xForceSimEnable AND Force_xTimeout THEN
	iAlarmID := 1005;
ELSE
	iAlarmID := 0;
END_IF;

HMI_iAutoStepShow := iAutoStep;
HMI_xLampEStop := xEStopLatched OR NOT HMI_xEStop;
HMI_xLampEnableOk := Dev_xRun;
HMI_xLampFault := xFaultAggregate;
HMI_iAlarmShow := iAlarmID;

StopLamp := Dev_xStop;
StartLamp := Dev_xRun;

          
END_PROGRAM

FUNCTION_BLOCK FB_Servo
  VAR_INPUT
    xEnable : BOOL;
    xJogPos : BOOL;
    xJogNeg : BOOL;
    xStop : BOOL;
    xResetFault : BOOL;
    xHome : BOOL;
    xUseVelCmd : BOOL;
    rVelCmd : REAL;
    rJogVel : REAL;
    rAcc : REAL;
    rDec : REAL;
  END_VAR
  VAR_OUTPUT
    xPowered : BOOL;
    xMoving : BOOL;
    xStandstill : BOOL;
    xHomed : BOOL;
    xFault : BOOL;
    rActPos : LREAL;
  END_VAR
  VAR_IN_OUT
    Axis : AXIS_REF_SM3;
  END_VAR
  VAR
    fbPower : MC_Power;
    fbJog : MC_MoveVelocity;
    fbStop : MC_Stop;
    fbHome : MC_Home;
    fbReset : MC_Reset;
    fbReadStatus : MC_ReadStatus;
    fbReadPos : MC_ReadActualPosition;
    xEnInternal : BOOL;
    fbSetPos : MC_SetPosition;
    xHomePrev : BOOL;
    xZeroReq : BOOL;
  END_VAR

            (* 读轴状态 / 实际位置 *)
fbReadStatus(Axis := Axis, Enable := TRUE);
fbReadPos(Axis := Axis, Enable := TRUE);

rActPos := fbReadPos.Position;
xStandstill := fbReadStatus.StandStill;
xMoving := fbReadStatus.DiscreteMotion OR fbReadStatus.ContinuousMotion;

(* 轴故障：仅 MC_ReadStatus.Errorstop，不用各 FB.Error *)
xFault := fbReadStatus.Errorstop;

(* 错误复位脉冲（来自停止钮长按 3s → AxisCmd_xResetFault） *)
fbReset(Axis := Axis, Execute := xResetFault);

(* 内部使能：请求使能且未停且非 Errorstop *)
xEnInternal := xEnable AND NOT xStop AND NOT fbReadStatus.Errorstop;

(* 功率级：Enable 恒 TRUE 以刷新；实际开/关看 bRegulatorOn/bDriveStart *)
fbPower(
	Axis := Axis,
	Enable := TRUE,
	bRegulatorOn := xEnInternal,
	bDriveStart := xEnInternal
);
(* Status=TRUE 表示轴可运动 *)
xPowered := fbPower.Status;

(* 回零上升沿：清除已回零，准备完成后置零 *)
IF xHome AND NOT xHomePrev THEN
	xHomed := FALSE;
	xZeroReq := FALSE;
END_IF;
xHomePrev := xHome;

(* ---------- 运动仲裁 ---------- *)
IF xStop OR NOT xEnable OR fbReadStatus.Errorstop THEN
	(* 停止 / 禁使能 / 故障：停速度指令并减速停 *)
	fbJog(Axis := Axis, Execute := FALSE);
	fbHome(Axis := Axis, Execute := FALSE, Position := 0.0);
	fbStop(Axis := Axis, Execute := TRUE, Deceleration := rDec);
	xZeroReq := FALSE;

ELSIF xHome THEN
	(* 回零：MC_Home Position:=0；完成后 MC_SetPosition 把当前点设为 0 *)
	fbStop(Axis := Axis, Execute := FALSE);
	fbJog(Axis := Axis, Execute := FALSE);
	fbHome(Axis := Axis, Execute := TRUE, Position := 0.0);
	IF fbHome.Done THEN
		xZeroReq := TRUE;
	END_IF;

ELSIF xUseVelCmd THEN
	(* 成对速度模式：使用有符号 rVelCmd（来自 FB_XDiff） *)
	fbStop(Axis := Axis, Execute := FALSE);
	fbHome(Axis := Axis, Execute := FALSE, Position := 0.0);
	IF ABS(rVelCmd) > 1.0E-6 AND xPowered THEN
		fbJog(Axis := Axis, Execute := TRUE, Velocity := rVelCmd, Acceleration := rAcc, Deceleration := rDec);
	ELSE
		fbJog(Axis := Axis, Execute := FALSE);
	END_IF;

ELSIF xJogPos XOR xJogNeg THEN
	(* 独立 JOG *)
	fbStop(Axis := Axis, Execute := FALSE);
	fbHome(Axis := Axis, Execute := FALSE, Position := 0.0);
	IF xPowered THEN
		IF xJogPos THEN
			fbJog(Axis := Axis, Execute := TRUE, Velocity := ABS(rJogVel), Acceleration := rAcc, Deceleration := rDec);
		ELSE
			fbJog(Axis := Axis, Execute := TRUE, Velocity := -ABS(rJogVel), Acceleration := rAcc, Deceleration := rDec);
		END_IF;
	ELSE
		fbJog(Axis := Axis, Execute := FALSE);
	END_IF;

ELSE
	(* 空闲 *)
	fbJog(Axis := Axis, Execute := FALSE);
	fbHome(Axis := Axis, Execute := FALSE, Position := 0.0);
	fbStop(Axis := Axis, Execute := FALSE);
END_IF;

(* 回零完成后：把当前位置设为坐标系 0 点 *)
fbSetPos(Axis := Axis, Execute := xZeroReq, Position := 0.0);
IF fbSetPos.Done THEN
	xHomed := TRUE;
	xZeroReq := FALSE;
END_IF;

          
END_FUNCTION_BLOCK

PROGRAM PRG_Force485
  VAR
    iSlaveStep : INT;
    iSlaveTry : INT;
    tonSlave : TON;
    wSnap : WORD;
    wRawLast : WORD;
    xTarePrev : BOOL;
    xUntarePrev : BOOL;
    xUnitInit : BOOL;
    diRaw : DINT;
    rTmp : REAL;
    xTareReq : BOOL;
  END_VAR

            (*==============================================================================
 * PRG_Force485 — SM1001 使能 + 发读等回文（最多3次）+ 去皮/换算
 *
 * 流程（严格按需求）：
 *   1) 使能 Modbus 从站 SM1001
 *   2) 发送一次读（破坏 Force_wInRaw 快照，等组态 FC03 通道写回 = 有回文）
 *   3) 有回文 → Force_xCommOk，进入成功态，不再重试
 *   4) 无回文 → 关闭 SM1001，重新使能，再读
 *   5) 3 次均无回文 → Force_xSlaveFail / 报警 1006
 *
 * 组态：读通道 FC03 0x0000 → Force_wInRaw（循环或由 Force_xReadTrig 触发均可）
 *============================================================================*)

Force_xTareDone := FALSE;

IF NOT Force_xEnable THEN
	SM1001 := FALSE;
	Force_xReadTrig := FALSE;
	Force_xCommOk := FALSE;
	Force_xTimeout := FALSE;
	Force_xTareBusy := FALSE;
	Force_xSlaveFail := FALSE;
	Force_iState := 0;
	iSlaveStep := 0;
	iSlaveTry := 0;
	RETURN;
END_IF;

CASE iSlaveStep OF
	0: (* 准备：先关从站，再进入使能 *)
		IF iSlaveTry >= 3 THEN
			SM1001 := FALSE;
			Force_xReadTrig := FALSE;
			Force_xSlaveFail := TRUE;
			Force_xTimeout := TRUE;
			Force_xCommOk := FALSE;
			Force_iState := -2;
			iSlaveStep := 99;
		ELSE
			SM1001 := FALSE;
			Force_xReadTrig := FALSE;
			Force_xCommOk := FALSE;
			tonSlave(IN := FALSE);
			tonSlave(IN := TRUE, PT := T#200MS);
			Force_iState := 0;
			iSlaveStep := 1;
		END_IF;

	1: (* 关断保持 *)
		SM1001 := FALSE;
		Force_xReadTrig := FALSE;
		tonSlave();
		IF tonSlave.Q THEN
			tonSlave(IN := FALSE);
			iSlaveStep := 2;
		END_IF;

	2: (* ① 使能从站 *)
		SM1001 := TRUE;
		Force_xReadTrig := FALSE;
		iSlaveTry := iSlaveTry + 1;
		tonSlave(IN := FALSE);
		tonSlave(IN := TRUE, PT := T#100MS);
		Force_iState := 1;
		iSlaveStep := 3;

	3: (* 使能稳定后：② 发读命令（破坏快照 + 读触发） *)
		SM1001 := TRUE;
		tonSlave();
		IF tonSlave.Q THEN
			(* 破坏映射值：有回文时通道会写回真实寄存器 *)
			wSnap := Force_wInRaw XOR 16#FFFF;
			Force_wInRaw := wSnap;
			Force_xReadTrig := FALSE;
			tonSlave(IN := FALSE);
			tonSlave(IN := TRUE, PT := T#20MS);
			Force_iState := 2;
			iSlaveStep := 4;
		END_IF;

	4: (* 读触发上升沿 *)
		SM1001 := TRUE;
		tonSlave();
		IF tonSlave.Q THEN
			Force_xReadTrig := TRUE;
			tonSlave(IN := FALSE);
			tonSlave(IN := TRUE, PT := T#500MS);
			Force_iState := 3;
			iSlaveStep := 5;
		END_IF;

	5: (* ③ 等回文：Force_wInRaw 被总线写回且不等于破坏值 *)
		SM1001 := TRUE;
		Force_xReadTrig := TRUE;
		tonSlave();
		IF Force_wInRaw <> wSnap THEN
			(* 有回文 → 成功，不再尝试 *)
			Force_xReadTrig := FALSE;
			Force_xCommOk := TRUE;
			Force_xTimeout := FALSE;
			Force_xSlaveFail := FALSE;
			wRawLast := Force_wInRaw;
			Force_iState := 4;
			tonSlave(IN := FALSE);
			iSlaveStep := 10;
		ELSIF tonSlave.Q THEN
			(* 无回文 → 关从站，回到 0 重新使能 *)
			Force_xReadTrig := FALSE;
			SM1001 := FALSE;
			Force_xCommOk := FALSE;
			Force_iState := 5;
			tonSlave(IN := FALSE);
			iSlaveStep := 0;
		END_IF;

	10: (* 成功：保持使能，不再重试使能 *)
		SM1001 := TRUE;
		Force_xReadTrig := FALSE;
		Force_xCommOk := TRUE;
		Force_xTimeout := FALSE;
		IF Force_wInRaw <> wRawLast THEN
			wRawLast := Force_wInRaw;
		END_IF;

	99: (* 3 次失败；复位清 Force_xSlaveFail 后从 0 重来 *)
		SM1001 := FALSE;
		Force_xReadTrig := FALSE;
		IF Force_xSlaveFail THEN
			Force_xTimeout := TRUE;
			Force_xCommOk := FALSE;
		ELSE
			iSlaveTry := 0;
			Force_xTimeout := FALSE;
			iSlaveStep := 0;
		END_IF;
END_CASE;

(* ----- 原始值换算（成功后持续；探测中也换算便于监视） ----- *)
diRaw := DWORD_TO_DINT(WORD_TO_DWORD(Force_wInRaw));
IF diRaw > 32767 THEN
	diRaw := diRaw - 65536;
END_IF;
Force_iRaw := DINT_TO_INT(diRaw);
IF Force_rScale < 1.0E-12 THEN
	rTmp := INT_TO_REAL(Force_iRaw);
ELSE
	rTmp := INT_TO_REAL(Force_iRaw) * Force_rScale;
END_IF;
IF NOT HMI_xForceSimEnable AND iSlaveStep = 10 THEN
	rForceAct := rTmp;
END_IF;

IF NOT xUnitInit AND iSlaveStep = 10 THEN
	Force_wOutUnit := 5;
	xUnitInit := TRUE;
END_IF;

xTareReq := FALSE;
IF iSlaveStep = 10 THEN
	IF ((HMI_xForceTare OR Tcp_xForceTare OR Logic_xForceTare) AND NOT xTarePrev) THEN
		Force_wOutTare := 1;
		xTareReq := TRUE;
		Force_xTareDone := TRUE;
	END_IF;
	xTarePrev := HMI_xForceTare OR Tcp_xForceTare OR Logic_xForceTare;
	IF Tcp_xForceTare THEN
		Tcp_xForceTare := FALSE;
	END_IF;
	IF Logic_xForceTare THEN
		Logic_xForceTare := FALSE;
	END_IF;

	IF ((HMI_xForceUntare OR Tcp_xForceUntare) AND NOT xUntarePrev) THEN
		Force_wOutTare := 2;
		xTareReq := TRUE;
		Force_xTareDone := TRUE;
	END_IF;
	xUntarePrev := HMI_xForceUntare OR Tcp_xForceUntare;
	IF Tcp_xForceUntare THEN
		Tcp_xForceUntare := FALSE;
	END_IF;
END_IF;

Force_xTareBusy := xTareReq;

          
END_PROGRAM

CONFIGURATION Device
END_CONFIGURATION

CONFIGURATION HIGH_SPEED_IO
END_CONFIGURATION

CONFIGURATION ETHERCAT
END_CONFIGURATION

CONFIGURATION MDX_EC
END_CONFIGURATION

CONFIGURATION Axis
END_CONFIGURATION

CONFIGURATION MDX_EC_1
END_CONFIGURATION

CONFIGURATION Axis_1
END_CONFIGURATION

CONFIGURATION MDX_EC_2
END_CONFIGURATION

CONFIGURATION Axis_2
END_CONFIGURATION

CONFIGURATION MDX_EC_3
END_CONFIGURATION

CONFIGURATION Axis_3
END_CONFIGURATION

CONFIGURATION MDX_EC_4
END_CONFIGURATION

CONFIGURATION Axis_4
END_CONFIGURATION

CONFIGURATION MODBUS_COM0
END_CONFIGURATION

CONFIGURATION modbus_protocol
END_CONFIGURATION
